(* IEC 61131-3 sources: Lasal/CPU_5344_V01/Class/CanTrend, 1 file *)

(* ---- CanTrend.st ---- *)
(*!
<Class
	Name               = "CanTrend"
	Revision           = "0.2"
	RealtimeTask       = "false"
	CyclicTask         = "false"
	BackgroundTask     = "false"
	Sigmatek           = "false"
	OSInterface        = "false"
	HighPriority       = "false"
	Automatic          = "false"
	UpdateMode         = "Prescan"
	SharedCommandTable = "true"
	Objectsize         = "(296,120)">
	<Channels>
		<Server Name="CobId" Visualized="false" Initialize="false" WriteProtected="true" Retentive="false"/>
		<Server Name="Server0" Visualized="true" Initialize="false" WriteProtected="false" Retentive="false"/>
		<Client Name="cCircular" Required="false" Internal="false" Comment="0= Once, 1= continues trend"/>
		<Client Name="cSigmaID" Required="false" Internal="false" Comment="0= All ID&apos;s 1= No SigmaTek ID&apos;s ( 16#700.. 16#71F)"/>
		<Client Name="IrqCannel" Required="false" Internal="false"/>
	</Channels>
	<Dependencies>
		<Files>
			<File Path=".\Class\CanTrend\CanTrendGl.h" Include="false"/>
		</Files>
	</Dependencies>
</Class>
*)
CanTrend : CLASS
	TYPE
	  CanTrendStr : STRUCT  //! <Type Comment="Can object ( ID, Size and Data)" Name="CanTrendStr"/>
	    ID : HDINT;  //! <Type Comment="CAN ID of the message" Name="CanTrendStr.ID"/>
	    Size : DINT;  //! <Type Comment="The size of CAN data message" Name="CanTrendStr.Size"/>
	    Data : ARRAY [1..8] OF HSINT;  //! <Type Comment="The Data in CAN message" Name="CanTrendStr.Data"/>
	    TimeStamp : UDINT;  //! <Type Comment="The Time when object is recieved" Name="CanTrendStr.TimeStamp"/>
	  END_STRUCT;
	END_TYPE
  //Servers:
	Server0 	: SvrChCmd_DINT;
	CobId 	: SvrCh_HDINT;
  //Clients:
	IrqCannel 	: CltCh_DINT;
	cCircular 	: CltCh_DINT;
	cSigmaID 	: CltCh_DINT;
  //Variables:
		pRxData 	: ^CanObjStr;			//! <Variable Comment="Pointer CAN object" Name="pRxData"/>
		pTrend 	: ^CanTrendStr;			//! <Variable Comment="Pointer to CAN object in trend buffer" Name="pTrend"/>
		aCanTrend : ARRAY [0..cMaxCanTrend] OF CanTrendStr;

		IrqChannelOn 	: DINT;			//! <Variable Comment="IrqChannel is connected " Name="IrqChannelOn"/>
  //Functions:

	FUNCTION VIRTUAL GLOBAL Init;
				//! <Function Comment="[#ENGLISH]&#13;&#10;" Name="WriteObjPtr"/>
	FUNCTION VIRTUAL GLOBAL WriteObjPtr
		VAR_INPUT
			CanObj 	: ^CanObjStr;			//! <Variable Comment="Pointer to CAN object" Name="WriteObjPtr.CanObj"/>
		END_VAR
		VAR_OUTPUT
			Result 	: DINT;			//! <Variable Comment="-1= Unvalid pointer, 0&gt;= Ok." Name="WriteObjPtr.Result"/>
		END_VAR;

	FUNCTION TrendObj;

	FUNCTION VIRTUAL GLOBAL Server0::Write
		VAR_INPUT
			input (EAX) 	: DINT;
		END_VAR
		VAR_OUTPUT
			result (EAX) 	: DINT;
		END_VAR;
  //Tables:
	FUNCTION @STD
		VAR_OUTPUT
			ret_code	: CONFSTATES;
		END_VAR;
	FUNCTION GLOBAL TAB @CT_;
END_CLASS;

FUNCTION VIRTUAL GLOBAL CanTrend::Init

	IrqChannelOn	:= IsClientConnected( #IrqCannel);
	If IsClientConnected( #cCircular) Then
		cCircular	:= cCircular.Read();
	End_If;
	If IsClientConnected( #cSigmaID) Then
		cSigmaID	:= cSigmaID.Read();
	End_If;

END_FUNCTION //VIRTUAL GLOBAL CanTrend::Init

FUNCTION VIRTUAL GLOBAL CanTrend::Server0::Write
	VAR_INPUT
		input (EAX) 	: DINT;
	END_VAR
	VAR_OUTPUT
		result (EAX) 	: DINT;
	END_VAR

If Input<> 0 Then
	pRxData	:= Input$^CanObjStr;
	TrendObj();
	Result	:= 0;
Else
	Result	:= -1;
End_If;

END_FUNCTION //VIRTUAL GLOBAL CanTrend::Server0::Write
//[#ENGLISH]
//[>CanObj]Pointer to CAN object
//[<Result]-1= Unvalid pointer, 0>= Ok.
FUNCTION VIRTUAL GLOBAL CanTrend::WriteObjPtr
VAR_INPUT
	CanObj		: ^CanObjStr;
END_VAR
VAR_OUTPUT
	Result		: DINT;
END_VAR

If CanObj<> 0 Then
	pRxData	:= CanObj;
	TrendObj();
	Result	:= 0;
Else
	Result	:= -1;
End_If;

END_FUNCTION //VIRTUAL GLOBAL CanTrend::WriteObjPtr

FUNCTION  CanTrend::TrendObj
VAR
	i			: Dint;
	Size		: DINT;
END_VAR

	If IrqChannelOn Then
		IrqCannel.Write( pRxData$Dint);
	End_If;

	pTrend	:= #aCanTrend[Server0]$CanTrendStr;
	pTrend^.ID		:= pRxData^.ID;
  CobId := pRxData^.ID; //

	If pTrend^.ID< 16#700 | pTrend^.ID> 16#71F | cSigmaID= 0 Then

		pTrend^.Size		:= Size	:= pRxData^.Size;
		pTrend^.TimeStamp	:= Ops.tAbsolute;

		// In test mode clear all the not used data for read-a-billety
		Case Size Of
		0:
			// No DATA so Clear all
			pTrend^.Data[1]$Dint	:= 0;
			pTrend^.Data[5]$Dint	:= 0;;
		1..7:
			// Copy the DATA and clear the rest
			For i:= 1 to Size Do
				pTrend^.Data[i]	:= pRxData^.Data[i];
			End_For;
			For i:= (Size+ 1) to 8 Do
				pTrend^.Data[i]	:= 0;
			End_For;
		8:
			// Copy the DATA
			pTrend^.Data[1]$Dint	:= pRxData^.Data[1]$Dint;
			pTrend^.Data[5]$Dint	:= pRxData^.Data[5]$Dint;
		Else
			// Other options not posible so clear DATA and generate an ERROR
			// No DATA so Clear all
			pTrend^.Data[1]$Dint	:= 0;
			pTrend^.Data[5]$Dint	:= 0;
		End_Case;

		If Server0< cMaxCanTrend Then
			Server0 += 1;
		Else
			If cCircular= 1 Then
				Server0	:= 0;
			End_If;
		End_If;
	End_If;

END_FUNCTION // CanTrend::TrendObj
